{attribute 'GeneratedUsingTerminal: EK1100-0000-0018'}
{attribute addProperty BoxType "EK1100-0000-0018"}
{attribute addProperty Id "boxesEK1122boxesEK1122_B55A8AA2348A_0001_EJ5151_0000_0016EJ5151_905C5FD836A_0002_EL1262_0000_0002EL1262_0FA571DE40A_0003_EL1262_0000_0003EL1262_0FA571DE40A_0004_EL1262_0050_0002EL1262_0FA571DE40A_0005_EL1262_0050_0003EL1262_0FA571DE40A_0006_EL2262_0000_0001EL2262_79C970B117A_0007_EL2262_0000_0002EL2262_147DB6E135A_0008_EL2262_0000_0003EL2262_147DB6E135A_0009_EL2262_0000_0004EL2262_9619875D40A_0010_EL3681_0000_0017EL3681_02A14E6431A_0011_EL3681_0000_0018EL3681_0095B62C32A_0012_EL3681_0000_0019EL3681_0095B62C32A_0013_EL3681_0000_0020EL3681_0095B62C32A_0014_EL5101_0000_0000EL5101_127DF9F120A_0015_EL5151_0000_0016EL5151_84FDBA5C40A_0016_EL5151_0000_0017EL5151_9335462842A_0017_EL5151_0000_0018EL5151_9335462842A_0018_EL5151_0000_0019EL5151_9335462842A_0019_EL5151_0000_0020EL5151_905C5FD836A_0020_EL5151_0000_0025EL5151_905C5FD836A_0021_EL5151_0000_0026EL5151_905C5FD836A_0022_EL5151_0080_0016EL5151_4D0E77FC36A_0023_EL5151_0080_0017EL5151_905C5FD836A_0024_EL5151_0080_0018EL5151_905C5FD836A_0025_EL5151_0080_0019EL5151_905C5FD836A_0026_EL5151_0080_0020EL5151_905C5FD836A_0027_EL5151_0080_0021EL5151_905C5FD836A_0028_EL3773_0000_0016EL3773_D0D76902198A_0029_EM7004_0000_9995EM7004_866015E192A_0041_AX8108_0100_0101AX8108_8297A621113A_0042_AX8108_0100_0102AX8108_F7A82895113A_0043_AX8108_0100_0103AX8108_F7A82895113A_0044_AX8108_0100_0104AX8108_F7A82895113A_0045_AX8108_0110_0102AX8108_F7A82895113A_0046_AX8108_0110_0103AX8108_F7A82895113A_0047_AX8108_0110_0104AX8108_F7A82895113A_0048_AX8108_0200_0103AX8108_F7A82895113A_0049_AX8108_0200_0104AX8108_F7A82895113A_0050_AX8108_0210_0103AX8108_F7A82895113A_0051_AX8108_0210_0104AX8108_F7A82895113A_0052_AX8118_0100_0101AX8118_8297A621113A_0053_AX8118_0100_0102AX8118_F7A82895113A_0054_AX8118_0100_0103AX8118_F7A82895113A_0055_AX8118_0100_0104AX8118_F7A82895113A_0056_AX8118_0110_0102AX8118_F7A82895113A_0057_AX8118_0110_0103AX8118_F7A82895113A_0058_AX8118_0110_0104AX8118_F7A82895113A_0059_AX8118_0200_0103AX8118_F7A82895113A_0060_AX8118_0200_0104AX8118_F7A82895113A_0061_AX8118_0210_0103AX8118_F7A82895113A_0062_AX8118_0210_0104AX8118_F7A82895113A_0063_AX8206_0100_0101AX8206_63F473B4136A_0064_AX8206_0100_0102AX8206_FA9FF81E136A_0065_AX8206_0100_0103AX8206_FA9FF81E136A_0066_AX8206_0100_0104AX8206_FA9FF81E136A_0067_AX8206_0110_0102AX8206_FA9FF81E136A_0068_AX8206_0110_0103AX8206_FA9FF81E136A_0069_AX8206_0110_0104AX8206_FA9FF81E136A_0070_AX8206_0200_0103AX8206_FA9FF81E136A_0071_AX8206_0200_0104AX8206_FA9FF81E136A_0072_AX8206_0210_0103AX8206_FA9FF81E136A_0073_AX8206_0210_0104AX8206_FA9FF81E136A_0074_EM7004_0000_9995EM7004_866015E192A_0075_AX8118_0100_0101AX8118_8297A621113"}
{attribute addProperty CRC "394885490"}
{attribute addProperty Size "5785"}
TYPE boxes_17897972 EXTENDS EK1100_1FC0878B :
STRUCT
	{attribute addProperty Name "boxesEK1122"}
	{attribute addProperty PreviousPort "boxes : B"}
	boxesEK1122 : boxesEK1122_B55A8AA2;
	{attribute addProperty Name "A_0001(EJ5151-0000-0016 )"}
	{attribute addProperty PreviousPort "boxesEK1122 : C"}
	A_0001_EJ5151_0000_0016 : EJ5151_905C5FD8;
	{attribute addProperty Name "A_0002(EL1262-0000-0002 )"}
	{attribute addProperty PreviousPort "A_0001(EJ5151-0000-0016 ) : B"}
	A_0002_EL1262_0000_0002 : EL1262_0FA571DE;
	{attribute addProperty Name "A_0003(EL1262-0000-0003 )"}
	{attribute addProperty PreviousPort "A_0002(EL1262-0000-0002 ) : B"}
	A_0003_EL1262_0000_0003 : EL1262_0FA571DE;
	{attribute addProperty Name "A_0004(EL1262-0050-0002 )"}
	{attribute addProperty PreviousPort "A_0003(EL1262-0000-0003 ) : B"}
	A_0004_EL1262_0050_0002 : EL1262_0FA571DE;
	{attribute addProperty Name "A_0005(EL1262-0050-0003 )"}
	{attribute addProperty PreviousPort "A_0004(EL1262-0050-0002 ) : B"}
	A_0005_EL1262_0050_0003 : EL1262_0FA571DE;
	{attribute addProperty Name "A_0006(EL2262-0000-0001 )"}
	{attribute addProperty PreviousPort "A_0005(EL1262-0050-0003 ) : B"}
	A_0006_EL2262_0000_0001 : EL2262_79C970B1;
	{attribute addProperty Name "A_0007(EL2262-0000-0002 )"}
	{attribute addProperty PreviousPort "A_0006(EL2262-0000-0001 ) : B"}
	A_0007_EL2262_0000_0002 : EL2262_147DB6E1;
	{attribute addProperty Name "A_0008(EL2262-0000-0003 )"}
	{attribute addProperty PreviousPort "A_0007(EL2262-0000-0002 ) : B"}
	A_0008_EL2262_0000_0003 : EL2262_147DB6E1;
	{attribute addProperty Name "A_0009(EL2262-0000-0004 )"}
	{attribute addProperty PreviousPort "A_0008(EL2262-0000-0003 ) : B"}
	A_0009_EL2262_0000_0004 : EL2262_9619875D;
	{attribute addProperty Name "A_0010(EL3681-0000-0017 )"}
	{attribute addProperty PreviousPort "A_0009(EL2262-0000-0004 ) : B"}
	A_0010_EL3681_0000_0017 : EL3681_02A14E64;
	{attribute addProperty Name "A_0011(EL3681-0000-0018 )"}
	{attribute addProperty PreviousPort "A_0010(EL3681-0000-0017 ) : B"}
	A_0011_EL3681_0000_0018 : EL3681_0095B62C;
	{attribute addProperty Name "A_0012(EL3681-0000-0019 )"}
	{attribute addProperty PreviousPort "A_0011(EL3681-0000-0018 ) : B"}
	A_0012_EL3681_0000_0019 : EL3681_0095B62C;
	{attribute addProperty Name "A_0013(EL3681-0000-0020 )"}
	{attribute addProperty PreviousPort "A_0012(EL3681-0000-0019 ) : B"}
	A_0013_EL3681_0000_0020 : EL3681_0095B62C;
	{attribute addProperty Name "A_0014(EL5101-0000-0000 )"}
	{attribute addProperty PreviousPort "A_0013(EL3681-0000-0020 ) : B"}
	A_0014_EL5101_0000_0000 : EL5101_127DF9F1;
	{attribute addProperty Name "A_0015(EL5151-0000-0016 )"}
	{attribute addProperty PreviousPort "A_0014(EL5101-0000-0000 ) : B"}
	A_0015_EL5151_0000_0016 : EL5151_84FDBA5C;
	{attribute addProperty Name "A_0016(EL5151-0000-0017 )"}
	{attribute addProperty PreviousPort "A_0015(EL5151-0000-0016 ) : B"}
	A_0016_EL5151_0000_0017 : EL5151_93354628;
	{attribute addProperty Name "A_0017(EL5151-0000-0018 )"}
	{attribute addProperty PreviousPort "A_0016(EL5151-0000-0017 ) : B"}
	A_0017_EL5151_0000_0018 : EL5151_93354628;
	{attribute addProperty Name "A_0018(EL5151-0000-0019 )"}
	{attribute addProperty PreviousPort "A_0017(EL5151-0000-0018 ) : B"}
	A_0018_EL5151_0000_0019 : EL5151_93354628;
	{attribute addProperty Name "A_0019(EL5151-0000-0020 )"}
	{attribute addProperty PreviousPort "A_0018(EL5151-0000-0019 ) : B"}
	A_0019_EL5151_0000_0020 : EL5151_905C5FD8;
	{attribute addProperty Name "A_0020(EL5151-0000-0025 )"}
	{attribute addProperty PreviousPort "A_0019(EL5151-0000-0020 ) : B"}
	A_0020_EL5151_0000_0025 : EL5151_905C5FD8;
	{attribute addProperty Name "A_0021(EL5151-0000-0026 )"}
	{attribute addProperty PreviousPort "A_0020(EL5151-0000-0025 ) : B"}
	A_0021_EL5151_0000_0026 : EL5151_905C5FD8;
	{attribute addProperty Name "A_0022(EL5151-0080-0016 )"}
	{attribute addProperty PreviousPort "A_0021(EL5151-0000-0026 ) : B"}
	A_0022_EL5151_0080_0016 : EL5151_4D0E77FC;
	{attribute addProperty Name "A_0023(EL5151-0080-0017 )"}
	{attribute addProperty PreviousPort "A_0022(EL5151-0080-0016 ) : B"}
	A_0023_EL5151_0080_0017 : EL5151_905C5FD8;
	{attribute addProperty Name "A_0024(EL5151-0080-0018 )"}
	{attribute addProperty PreviousPort "A_0023(EL5151-0080-0017 ) : B"}
	A_0024_EL5151_0080_0018 : EL5151_905C5FD8;
	{attribute addProperty Name "A_0025(EL5151-0080-0019 )"}
	{attribute addProperty PreviousPort "A_0024(EL5151-0080-0018 ) : B"}
	A_0025_EL5151_0080_0019 : EL5151_905C5FD8;
	{attribute addProperty Name "A_0026(EL5151-0080-0020 )"}
	{attribute addProperty PreviousPort "A_0025(EL5151-0080-0019 ) : B"}
	A_0026_EL5151_0080_0020 : EL5151_905C5FD8;
	{attribute addProperty Name "A_0027(EL5151-0080-0021 )"}
	{attribute addProperty PreviousPort "A_0026(EL5151-0080-0020 ) : B"}
	A_0027_EL5151_0080_0021 : EL5151_905C5FD8;
	{attribute addProperty Name "A_0028(EL3773-0000-0016 )"}
	{attribute addProperty PreviousPort "A_0027(EL5151-0080-0021 ) : B"}
	A_0028_EL3773_0000_0016 : EL3773_D0D76902;
	{attribute addProperty Name "A_0029(EM7004-0000-9995 )"}
	{attribute addProperty PreviousPort "A_0028(EL3773-0000-0016 ) : B"}
	A_0029_EM7004_0000_9995 : EM7004_866015E1;
	{attribute addProperty Name "A_0041(AX8108-0100-0101 )"}
	{attribute addProperty PreviousPort "A_0029(EM7004-0000-9995 ) : B"}
	A_0041_AX8108_0100_0101 : AX8108_8297A621;
	{attribute addProperty Name "A_0042(AX8108-0100-0102 )"}
	{attribute addProperty PreviousPort "A_0041(AX8108-0100-0101 ) : B"}
	A_0042_AX8108_0100_0102 : AX8108_F7A82895;
	{attribute addProperty Name "A_0043(AX8108-0100-0103 )"}
	{attribute addProperty PreviousPort "A_0042(AX8108-0100-0102 ) : B"}
	A_0043_AX8108_0100_0103 : AX8108_F7A82895;
	{attribute addProperty Name "A_0044(AX8108-0100-0104 )"}
	{attribute addProperty PreviousPort "A_0043(AX8108-0100-0103 ) : B"}
	A_0044_AX8108_0100_0104 : AX8108_F7A82895;
	{attribute addProperty Name "A_0045(AX8108-0110-0102 )"}
	{attribute addProperty PreviousPort "A_0044(AX8108-0100-0104 ) : B"}
	A_0045_AX8108_0110_0102 : AX8108_F7A82895;
	{attribute addProperty Name "A_0046(AX8108-0110-0103 )"}
	{attribute addProperty PreviousPort "A_0045(AX8108-0110-0102 ) : B"}
	A_0046_AX8108_0110_0103 : AX8108_F7A82895;
	{attribute addProperty Name "A_0047(AX8108-0110-0104 )"}
	{attribute addProperty PreviousPort "A_0046(AX8108-0110-0103 ) : B"}
	A_0047_AX8108_0110_0104 : AX8108_F7A82895;
	{attribute addProperty Name "A_0048(AX8108-0200-0103 )"}
	{attribute addProperty PreviousPort "A_0047(AX8108-0110-0104 ) : B"}
	A_0048_AX8108_0200_0103 : AX8108_F7A82895;
	{attribute addProperty Name "A_0049(AX8108-0200-0104 )"}
	{attribute addProperty PreviousPort "A_0048(AX8108-0200-0103 ) : B"}
	A_0049_AX8108_0200_0104 : AX8108_F7A82895;
	{attribute addProperty Name "A_0050(AX8108-0210-0103 )"}
	{attribute addProperty PreviousPort "A_0049(AX8108-0200-0104 ) : B"}
	A_0050_AX8108_0210_0103 : AX8108_F7A82895;
	{attribute addProperty Name "A_0051(AX8108-0210-0104 )"}
	{attribute addProperty PreviousPort "A_0050(AX8108-0210-0103 ) : B"}
	A_0051_AX8108_0210_0104 : AX8108_F7A82895;
	{attribute addProperty Name "A_0052(AX8118-0100-0101 )"}
	{attribute addProperty PreviousPort "A_0051(AX8108-0210-0104 ) : B"}
	A_0052_AX8118_0100_0101 : AX8118_8297A621;
	{attribute addProperty Name "A_0053(AX8118-0100-0102 )"}
	{attribute addProperty PreviousPort "A_0052(AX8118-0100-0101 ) : B"}
	A_0053_AX8118_0100_0102 : AX8118_F7A82895;
	{attribute addProperty Name "A_0054(AX8118-0100-0103 )"}
	{attribute addProperty PreviousPort "A_0053(AX8118-0100-0102 ) : B"}
	A_0054_AX8118_0100_0103 : AX8118_F7A82895;
	{attribute addProperty Name "A_0055(AX8118-0100-0104 )"}
	{attribute addProperty PreviousPort "A_0054(AX8118-0100-0103 ) : B"}
	A_0055_AX8118_0100_0104 : AX8118_F7A82895;
	{attribute addProperty Name "A_0056(AX8118-0110-0102 )"}
	{attribute addProperty PreviousPort "A_0055(AX8118-0100-0104 ) : B"}
	A_0056_AX8118_0110_0102 : AX8118_F7A82895;
	{attribute addProperty Name "A_0057(AX8118-0110-0103 )"}
	{attribute addProperty PreviousPort "A_0056(AX8118-0110-0102 ) : B"}
	A_0057_AX8118_0110_0103 : AX8118_F7A82895;
	{attribute addProperty Name "A_0058(AX8118-0110-0104 )"}
	{attribute addProperty PreviousPort "A_0057(AX8118-0110-0103 ) : B"}
	A_0058_AX8118_0110_0104 : AX8118_F7A82895;
	{attribute addProperty Name "A_0059(AX8118-0200-0103 )"}
	{attribute addProperty PreviousPort "A_0058(AX8118-0110-0104 ) : B"}
	A_0059_AX8118_0200_0103 : AX8118_F7A82895;
	{attribute addProperty Name "A_0060(AX8118-0200-0104 )"}
	{attribute addProperty PreviousPort "A_0059(AX8118-0200-0103 ) : B"}
	A_0060_AX8118_0200_0104 : AX8118_F7A82895;
	{attribute addProperty Name "A_0061(AX8118-0210-0103 )"}
	{attribute addProperty PreviousPort "A_0060(AX8118-0200-0104 ) : B"}
	A_0061_AX8118_0210_0103 : AX8118_F7A82895;
	{attribute addProperty Name "A_0062(AX8118-0210-0104 )"}
	{attribute addProperty PreviousPort "A_0061(AX8118-0210-0103 ) : B"}
	A_0062_AX8118_0210_0104 : AX8118_F7A82895;
	{attribute addProperty Name "A_0063(AX8206-0100-0101 )"}
	{attribute addProperty PreviousPort "A_0062(AX8118-0210-0104 ) : B"}
	A_0063_AX8206_0100_0101 : AX8206_63F473B4;
	{attribute addProperty Name "A_0064(AX8206-0100-0102 )"}
	{attribute addProperty PreviousPort "A_0063(AX8206-0100-0101 ) : B"}
	A_0064_AX8206_0100_0102 : AX8206_FA9FF81E;
	{attribute addProperty Name "A_0065(AX8206-0100-0103 )"}
	{attribute addProperty PreviousPort "A_0064(AX8206-0100-0102 ) : B"}
	A_0065_AX8206_0100_0103 : AX8206_FA9FF81E;
	{attribute addProperty Name "A_0066(AX8206-0100-0104 )"}
	{attribute addProperty PreviousPort "A_0065(AX8206-0100-0103 ) : B"}
	A_0066_AX8206_0100_0104 : AX8206_FA9FF81E;
	{attribute addProperty Name "A_0067(AX8206-0110-0102 )"}
	{attribute addProperty PreviousPort "A_0066(AX8206-0100-0104 ) : B"}
	A_0067_AX8206_0110_0102 : AX8206_FA9FF81E;
	{attribute addProperty Name "A_0068(AX8206-0110-0103 )"}
	{attribute addProperty PreviousPort "A_0067(AX8206-0110-0102 ) : B"}
	A_0068_AX8206_0110_0103 : AX8206_FA9FF81E;
	{attribute addProperty Name "A_0069(AX8206-0110-0104 )"}
	{attribute addProperty PreviousPort "A_0068(AX8206-0110-0103 ) : B"}
	A_0069_AX8206_0110_0104 : AX8206_FA9FF81E;
	{attribute addProperty Name "A_0070(AX8206-0200-0103 )"}
	{attribute addProperty PreviousPort "A_0069(AX8206-0110-0104 ) : B"}
	A_0070_AX8206_0200_0103 : AX8206_FA9FF81E;
	{attribute addProperty Name "A_0071(AX8206-0200-0104 )"}
	{attribute addProperty PreviousPort "A_0070(AX8206-0200-0103 ) : B"}
	A_0071_AX8206_0200_0104 : AX8206_FA9FF81E;
	{attribute addProperty Name "A_0072(AX8206-0210-0103 )"}
	{attribute addProperty PreviousPort "A_0071(AX8206-0200-0104 ) : B"}
	A_0072_AX8206_0210_0103 : AX8206_FA9FF81E;
	{attribute addProperty Name "A_0073(AX8206-0210-0104 )"}
	{attribute addProperty PreviousPort "A_0072(AX8206-0210-0103 ) : B"}
	A_0073_AX8206_0210_0104 : AX8206_FA9FF81E;
	{attribute addProperty Name "A_0074(EM7004-0000-9995)"}
	{attribute addProperty PreviousPort "A_0073(AX8206-0210-0104 ) : B"}
	A_0074_EM7004_0000_9995 : EM7004_866015E1;
	{attribute addProperty Name "A_0075(AX8118-0100-0101)"}
	{attribute addProperty PreviousPort "A_0074(EM7004-0000-9995) : B"}
	A_0075_AX8118_0100_0101 : AX8118_8297A621;
END_STRUCT
END_TYPE

(* stored: Version 1.2.0.0, ProductVersion 3.1.4024.11
   DUT boxes_17897972: Id {8bf135f8-905a-4fe7-ace2-9404984ace5a} *)
